// TIA Portal V16 export
// export: Created 2022-09-01T13:36:50.8725323Z, ExportSetting WithDefaults, DisplayName Totally Integrated Automation Portal, DisplayVersion V16, DisplayName TIA Portal Version Control Interface, DisplayVersion V16, DisplayName TIA Portal Openness, DisplayVersion V16, DisplayName STEP 7 Professional, DisplayVersion V16, DisplayName STEP 7 Safety, DisplayVersion V16, DisplayName WinCC Advanced, DisplayVersion V16
FUNCTION "Alarmes_Disparos_1" : Void   // FC22, LAD
{ S7_Optimized_Access := 'TRUE' }
VERSION : 0.1
// stored: AutoNumber true, IsIECCheckEnabled false, SetENOAutomatically false, UDAEnableTagReadback false
   VAR_TEMP   // added for the SCL form of the ladder/FBD networks
      _w1 : Bool;
      _w2 : Bool;
      _w3 : Bool;
      _w4 : Bool;
      _w5 : Bool;
      _w6 : Bool;
      _w7 : Bool;
      _w8 : Bool;
      _w9 : Bool;
      _w10 : Bool;
      _w11 : Bool;
      _w12 : Bool;
      _w13 : Bool;
      _w14 : Bool;
      _w15 : Bool;
      _w16 : Bool;
      _w17 : Bool;
      _w18 : Bool;
      _w19 : Bool;
      _w20 : Bool;
      _w21 : Bool;
      _w22 : Bool;
   END_VAR
BEGIN

REGION Network 1: Ativa contacto de alarme disparos para alarme luminoso
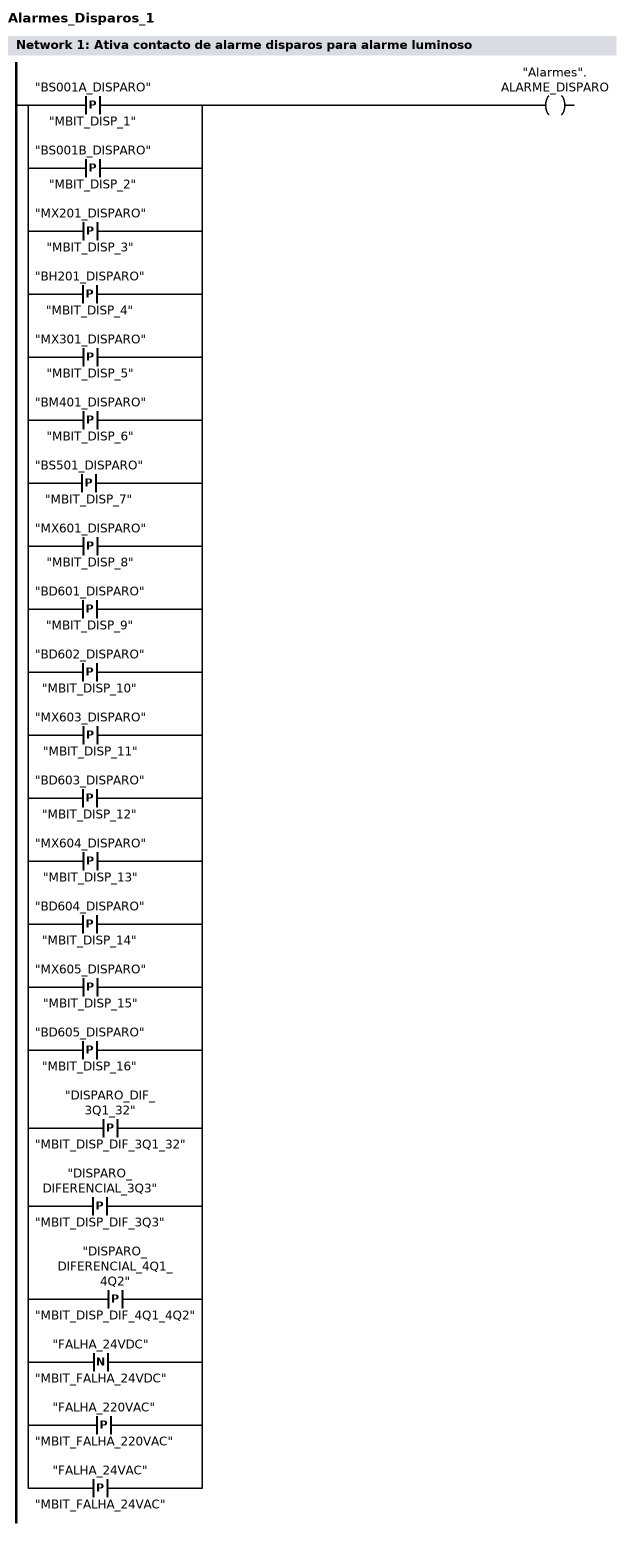
   RUNG wire#powerrail
      P_Contact(operand := "BS001A_DISPARO", bit := "MBIT_DISP_1")
      wire#w1
      Coil( "Alarmes".ALARME_DISPARO )
   END_RUNG
   RUNG wire#powerrail
      P_Contact(operand := "BS001B_DISPARO", bit := "MBIT_DISP_2")
   END_RUNG wire#w1
   RUNG wire#powerrail
      P_Contact(operand := "MX201_DISPARO", bit := "MBIT_DISP_3")
   END_RUNG wire#w1
   RUNG wire#powerrail
      P_Contact(operand := "BH201_DISPARO", bit := "MBIT_DISP_4")
   END_RUNG wire#w1
   RUNG wire#powerrail
      P_Contact(operand := "MX301_DISPARO", bit := "MBIT_DISP_5")
   END_RUNG wire#w1
   RUNG wire#powerrail
      P_Contact(operand := "BM401_DISPARO", bit := "MBIT_DISP_6")
   END_RUNG wire#w1
   RUNG wire#powerrail
      P_Contact(operand := "BS501_DISPARO", bit := "MBIT_DISP_7")
   END_RUNG wire#w1
   RUNG wire#powerrail
      P_Contact(operand := "MX601_DISPARO", bit := "MBIT_DISP_8")
   END_RUNG wire#w1
   RUNG wire#powerrail
      P_Contact(operand := "BD601_DISPARO", bit := "MBIT_DISP_9")
   END_RUNG wire#w1
   RUNG wire#powerrail
      P_Contact(operand := "BD602_DISPARO", bit := "MBIT_DISP_10")
   END_RUNG wire#w1
   RUNG wire#powerrail
      P_Contact(operand := "MX603_DISPARO", bit := "MBIT_DISP_11")
   END_RUNG wire#w1
   RUNG wire#powerrail
      P_Contact(operand := "BD603_DISPARO", bit := "MBIT_DISP_12")
   END_RUNG wire#w1
   RUNG wire#powerrail
      P_Contact(operand := "MX604_DISPARO", bit := "MBIT_DISP_13")
   END_RUNG wire#w1
   RUNG wire#powerrail
      P_Contact(operand := "BD604_DISPARO", bit := "MBIT_DISP_14")
   END_RUNG wire#w1
   RUNG wire#powerrail
      P_Contact(operand := "MX605_DISPARO", bit := "MBIT_DISP_15")
   END_RUNG wire#w1
   RUNG wire#powerrail
      P_Contact(operand := "BD605_DISPARO", bit := "MBIT_DISP_16")
   END_RUNG wire#w1
   RUNG wire#powerrail
      P_Contact(operand := "DISPARO_DIF_3Q1_32", bit := "MBIT_DISP_DIF_3Q1_32")
   END_RUNG wire#w1
   RUNG wire#powerrail
      P_Contact(operand := "DISPARO_DIFERENCIAL_3Q3", bit := "MBIT_DISP_DIF_3Q3")
   END_RUNG wire#w1
   RUNG wire#powerrail
      P_Contact(operand := "DISPARO_DIFERENCIAL_4Q1_4Q2", bit := "MBIT_DISP_DIF_4Q1_4Q2")
   END_RUNG wire#w1
   RUNG wire#powerrail
      N_Contact(operand := "FALHA_24VDC", bit := "MBIT_FALHA_24VDC")
   END_RUNG wire#w1
   RUNG wire#powerrail
      P_Contact(operand := "FALHA_220VAC", bit := "MBIT_FALHA_220VAC")
   END_RUNG wire#w1
   RUNG wire#powerrail
      P_Contact(operand := "FALHA_24VAC", bit := "MBIT_FALHA_24VAC")
   END_RUNG wire#w1
   // the same network as SCL:
   #_w1 := "BS001A_DISPARO" AND NOT "MBIT_DISP_1";   // rising edge of "BS001A_DISPARO"
   "MBIT_DISP_1" := "BS001A_DISPARO";
   #_w2 := "BS001B_DISPARO" AND NOT "MBIT_DISP_2";   // rising edge of "BS001B_DISPARO"
   "MBIT_DISP_2" := "BS001B_DISPARO";
   #_w3 := "MX201_DISPARO" AND NOT "MBIT_DISP_3";   // rising edge of "MX201_DISPARO"
   "MBIT_DISP_3" := "MX201_DISPARO";
   #_w4 := "BH201_DISPARO" AND NOT "MBIT_DISP_4";   // rising edge of "BH201_DISPARO"
   "MBIT_DISP_4" := "BH201_DISPARO";
   #_w5 := "MX301_DISPARO" AND NOT "MBIT_DISP_5";   // rising edge of "MX301_DISPARO"
   "MBIT_DISP_5" := "MX301_DISPARO";
   #_w6 := "BM401_DISPARO" AND NOT "MBIT_DISP_6";   // rising edge of "BM401_DISPARO"
   "MBIT_DISP_6" := "BM401_DISPARO";
   #_w7 := "BS501_DISPARO" AND NOT "MBIT_DISP_7";   // rising edge of "BS501_DISPARO"
   "MBIT_DISP_7" := "BS501_DISPARO";
   #_w8 := "MX601_DISPARO" AND NOT "MBIT_DISP_8";   // rising edge of "MX601_DISPARO"
   "MBIT_DISP_8" := "MX601_DISPARO";
   #_w9 := "BD601_DISPARO" AND NOT "MBIT_DISP_9";   // rising edge of "BD601_DISPARO"
   "MBIT_DISP_9" := "BD601_DISPARO";
   #_w10 := "BD602_DISPARO" AND NOT "MBIT_DISP_10";   // rising edge of "BD602_DISPARO"
   "MBIT_DISP_10" := "BD602_DISPARO";
   #_w11 := "MX603_DISPARO" AND NOT "MBIT_DISP_11";   // rising edge of "MX603_DISPARO"
   "MBIT_DISP_11" := "MX603_DISPARO";
   #_w12 := "BD603_DISPARO" AND NOT "MBIT_DISP_12";   // rising edge of "BD603_DISPARO"
   "MBIT_DISP_12" := "BD603_DISPARO";
   #_w13 := "MX604_DISPARO" AND NOT "MBIT_DISP_13";   // rising edge of "MX604_DISPARO"
   "MBIT_DISP_13" := "MX604_DISPARO";
   #_w14 := "BD604_DISPARO" AND NOT "MBIT_DISP_14";   // rising edge of "BD604_DISPARO"
   "MBIT_DISP_14" := "BD604_DISPARO";
   #_w15 := "MX605_DISPARO" AND NOT "MBIT_DISP_15";   // rising edge of "MX605_DISPARO"
   "MBIT_DISP_15" := "MX605_DISPARO";
   #_w16 := "BD605_DISPARO" AND NOT "MBIT_DISP_16";   // rising edge of "BD605_DISPARO"
   "MBIT_DISP_16" := "BD605_DISPARO";
   #_w17 := "DISPARO_DIF_3Q1_32" AND NOT "MBIT_DISP_DIF_3Q1_32";   // rising edge of "DISPARO_DIF_3Q1_32"
   "MBIT_DISP_DIF_3Q1_32" := "DISPARO_DIF_3Q1_32";
   #_w18 := "DISPARO_DIFERENCIAL_3Q3" AND NOT "MBIT_DISP_DIF_3Q3";   // rising edge of "DISPARO_DIFERENCIAL_3Q3"
   "MBIT_DISP_DIF_3Q3" := "DISPARO_DIFERENCIAL_3Q3";
   #_w19 := "DISPARO_DIFERENCIAL_4Q1_4Q2" AND NOT "MBIT_DISP_DIF_4Q1_4Q2";   // rising edge of "DISPARO_DIFERENCIAL_4Q1_4Q2"
   "MBIT_DISP_DIF_4Q1_4Q2" := "DISPARO_DIFERENCIAL_4Q1_4Q2";
   #_w20 := NOT "FALHA_24VDC" AND "MBIT_FALHA_24VDC";   // falling edge of "FALHA_24VDC"
   "MBIT_FALHA_24VDC" := "FALHA_24VDC";
   #_w21 := "FALHA_220VAC" AND NOT "MBIT_FALHA_220VAC";   // rising edge of "FALHA_220VAC"
   "MBIT_FALHA_220VAC" := "FALHA_220VAC";
   #_w22 := "FALHA_24VAC" AND NOT "MBIT_FALHA_24VAC";   // rising edge of "FALHA_24VAC"
   "MBIT_FALHA_24VAC" := "FALHA_24VAC";
   "Alarmes".ALARME_DISPARO := #_w1 OR #_w2 OR #_w3 OR #_w4 OR #_w5 OR #_w6 OR #_w7 OR #_w8 OR #_w9 OR #_w10 OR #_w11 OR #_w12 OR #_w13 OR #_w14 OR #_w15 OR #_w16 OR #_w17 OR #_w18 OR #_w19 OR #_w20 OR #_w21 OR #_w22;
END_REGION
END_FUNCTION
